	_nBufferIdx:= _nBufferIdx + 1;
	IF _nBufferIdx >= 3 THEN
		_nBufferIdx:= 1;
	END_IF

	CASE _nBufferIdx OF
		1:
			_pWriteBuffer:= _pBuffer1;
			_pReadBuffer:= _pBuffer2;

			_pWriteBufferTime:= ADR(_aBufferTime1);
			_pReadBufferTime:= ADR(_aBufferTime2);
		2:
			_pWriteBuffer:= _pBuffer2;
			_pReadBuffer:= _pBuffer1;

			_pWriteBufferTime:= ADR(_aBufferTime2);
			_pReadBufferTime:= ADR(_aBufferTime1);
	END_CASE

	nElements:= _nBufferEntry_Add;

	_nBufferEntry_Add:= 0;
	_bLock:= FALSE;
END_IF
END_METHOD

METHOD AddData : BOOL
VAR_INPUT
	pDataIn: PVOID;
END_VAR
VAR
END_VAR
IF TestAndSet(_bLock) THEN

	IF _pWriteBuffer <> 0 AND pDataIn <> 0 THEN

		IF _nBufferEntry_Add >= cEntryCount THEN
			_nBufferEntry_Add:= cEntryCount - 1;
		END_IF

		MEMCPY(_pWriteBuffer + (_nBufferEntry_Add * _nDataSize), pDataIn, _nDataSize);

		_nBufferEntry_Add:= _nBufferEntry_Add + 1;

		IF _pWriteBufferTime <> 0 THEN
			_pWriteBufferTime^[_nBufferEntry_Add]:= F_GetActualDcTime64();
		END_IF

	END_IF

	_bLock:= FALSE;
END_IF
END_METHOD

METHOD GetData : BOOL
VAR_INPUT
	nElement: UDINT(1..cEntryCount);
	pDataOut: PVOID;
END_VAR
VAR
END_VAR
IF nElement <= nElements THEN
	IF pDataOut <> 0 AND _pReadBuffer <> 0 THEN
		MEMCPY(pDataOut, _pReadBuffer + ((nElement-1) * _nDataSize), _nDataSize);
	END_IF
END_IF
END_METHOD

METHOD GetTimestamp : ULINT
VAR_INPUT
	nElement: UDINT(1..cEntryCount);
END_VAR
VAR
END_VAR
IF _pReadBufferTime <> 0 THEN
	GetTimestamp:= _pReadBufferTime^[nElement];
END_IF
END_METHOD

END_FUNCTION_BLOCK

// ---- POUs/Analytics/[Helper]/FB_GetSampleIndex.TcPOU
FUNCTION_BLOCK FB_GetSampleIndex
VAR_INPUT
	nSample: UDINT;
	nOverSamplingFactor: UDINT;
	nMaxOverSampling: UDINT;
	nTimestamp: ULINT;
END_VAR
VAR_OUTPUT
	bNewIndex: BOOL;
	nIndex: UDINT;
END_VAR
VAR
	nIndexFactor: UDINT;
	nLastIndex: UDINT;
	nLastTimestamp: ULINT;
END_VAR


nIndex:= 1;

IF nOverSamplingFactor > 0 THEN
	nIndexFactor:= nMaxOverSampling / nOverSamplingFactor;

	IF nIndexFactor > 0 THEN
		nIndex:= (nSample - 1) / nIndexFactor;
		nIndex:= nIndex + 1;
	END_IF

	IF nIndex > nOverSamplingFactor THEN
		nIndex:= nOverSamplingFactor;
	END_IF
END_IF

bNewIndex:= nIndex <> nLastIndex OR nLastTimestamp <> nTimestamp;

nLastIndex:= nIndex;
nLastTimestamp:= nTimestamp;

END_FUNCTION_BLOCK

// ---- POUs/Analytics/[Helper]/F_AlyTimestampToFileTime.TcPOU
FUNCTION F_AlyTimestampToFileTime : ULINT
VAR_INPUT
	tTimestamp: ULINT;
END_VAR
VAR
	tFileTime: T_FILETIME;
	
	fbToUTC: FB_TzSpecificLocalTimeToFileTime;
	//W. Europe Daylight Time
	//(UTC+01:00) Amsterdam, Berlin, Bern, Rome, Stockholm, Vienna
	tzInfo: ST_TimeZoneInformation := (bias := -60, standardDate := (wMonth := 10 ,wDay:=5, wHour := 3), daylightDate := (wMonth := 3, wDay:=5, wHour := 2), daylightBias := -60);
END_VAR

tFileTime:= DCTIME64_TO_Filetime(tTimestamp);

fbToUTC(in:= tFileTime, tzInfo:= tzInfo);
F_AlyTimestampToFileTime:= ULARGE_TO_ULINT(ULARGE_INTEGER(fbToUTC.out.dwHighDateTime, fbToUTC.out.dwLowDateTime));

END_FUNCTION

// ---- POUs/Analytics/[Helper]/F_AlyTimestampToLocalTime.TcPOU
FUNCTION F_AlyTimestampToLocalTime : ULINT
VAR_INPUT
	tTimestamp: ULINT;
END_VAR
VAR
	tFileTime: T_FILETIME;
END_VAR

tFileTime:= DCTIME64_TO_Filetime(tTimestamp);
F_AlyTimestampToLocalTime:= ULARGE_TO_ULINT(ULARGE_INTEGER(tFileTime.dwHighDateTime, tFileTime.dwLowDateTime));

END_FUNCTION

// ---- POUs/Analytics/[Helper]/F_ANY_Negation.TcPOU
FUNCTION F_ANY_Negation : BOOL
VAR_INPUT
	Input: ANY;
END_VAR
VAR
	bReturn: BOOL;
	pREAL: POINTER TO REAL;
	pLREAL: POINTER TO LREAL;
	pBOOL: POINTER TO BOOL;
	pBYTE: POINTER TO BYTE;
	pINT: POINTER TO INT;
	pDINT: POINTER TO DINT;
	pLINT: POINTER TO LINT;
	pUINT: POINTER TO UINT;
	pUDINT: POINTER TO UDINT;
	pULINT: POINTER TO ULINT;
	pWORD: POINTER TO WORD;
	pDWORD: POINTER TO DWORD;
	pLWORD: POINTER TO LWORD;
END_VAR

IF input.pValue <> 0 THEN
	bReturn:= TRUE;

	CASE Input.TypeClass OF
		__SYSTEM.TYPE_CLASS.TYPE_REAL:
			pREAL:= input.pValue;
			pREAL^:= pREAL^ * -1;
		__SYSTEM.TYPE_CLASS.TYPE_LREAL:
			pLREAL:= input.pValue;
			pLREAL^:= pLREAL^ * -1;
		__SYSTEM.TYPE_CLASS.TYPE_BOOL:
			pBOOL:= input.pValue;
			pBOOL^:= NOT pBOOL^;
		__SYSTEM.TYPE_CLASS.TYPE_BYTE:
			pBYTE:= input.pValue;
			pBYTE^:= NOT pBYTE^;
		__SYSTEM.TYPE_CLASS.TYPE_INT:
			pINT:= input.pValue;
			pINT^:= pINT^ * -1;
		__SYSTEM.TYPE_CLASS.TYPE_DINT:
			pDINT:= input.pValue;
			pDINT^:= pDINT^ * -1;
		__SYSTEM.TYPE_CLASS.TYPE_LINT:
			pLINT:= input.pValue;
			pLINT^:= pLINT^ * -1;
		__SYSTEM.TYPE_CLASS.TYPE_UINT:
			pUINT:= input.pValue;
			pUINT^:= NOT pUINT^;
		__SYSTEM.TYPE_CLASS.TYPE_UDINT:
			pUDINT:= input.pValue;
			pUDINT^:= NOT pUDINT^;
		__SYSTEM.TYPE_CLASS.TYPE_ULINT:
			pULINT:= input.pValue;
			pULINT^:= NOT pULINT^;
		__SYSTEM.TYPE_CLASS.TYPE_WORD:
			pWORD:= input.pValue;
			pWORD^:= NOT pWORD^;
		__SYSTEM.TYPE_CLASS.TYPE_DWORD:
			pDWORD:= input.pValue;
			pDWORD^:= NOT pDWORD^;
		__SYSTEM.TYPE_CLASS.TYPE_LWORD:
			pLWORD:= input.pValue;
			pLWORD^:= NOT pLWORD^;
		ELSE
			bReturn:= FALSE;
	END_CASE
END_IF

F_ANY_Negation:= bReturn;

END_FUNCTION

// ---- POUs/Analytics/[Helper]/F_ARRAY_To_LREAL_ARRAY.TcPOU
FUNCTION F_ARRAY_To_LREAL_ARRAY : BOOL
VAR_INPUT
	pDataIn: POINTER TO BYTE;
	cbDataIn: UDINT;
	eDataType: E_DTType;
END_VAR
VAR_IN_OUT
	aDataOut: ARRAY [*] OF LREAL;
END_VAR
VAR
	i: DINT;
	nPos: UDINT;
	
	pBOOL: POINTER TO BOOL;
	pBYTE: POINTER TO BYTE;
	pWORD: POINTER TO WORD;
	pDWORD: POINTER TO DWORD;
	pSINT: POINTER TO SINT;
	pUSINT: POINTER TO USINT;
	pINT: POINTER TO INT;
	pUINT: POINTER TO UINT;
	pDINT: POINTER TO DINT;
	pUDINT: POINTER TO UDINT;
	pLINT: POINTER TO LINT;
	pULINT: POINTER TO ULINT;
	pREAL: POINTER TO REAL;
	pLREAL: POINTER TO LREAL;
	pLWORD: POINTER TO LWORD;
END_VAR

FOR i := LOWER_BOUND(aDataOut,1) TO UPPER_BOUND(aDataOut,1) DO
	CASE eDataType OF
		E_DTType.NotInitialized:
			F_ARRAY_To_LREAL_ARRAY:= FALSE;
			RETURN;
		E_DTType.BOOL_:
			IF (nPos * 1) < cbDataIn THEN
				pBOOL:= pDataIn + (nPos * 1);
				aDataOut[i] := TO_LREAL(pBOOL^);
			END_IF
		E_DTType.BYTE_:
			IF (nPos * 1) < cbDataIn THEN
				pBYTE:= pDataIn + (nPos * 1);
				aDataOut[i] := TO_LREAL(pBYTE^);
			END_IF
		E_DTType.WORD_:
			IF (nPos * 2) < cbDataIn THEN
				pWORD:= pDataIn + (nPos * 2);
				aDataOut[i] := TO_LREAL(pWORD^);
			END_IF
		E_DTType.DWORD_:
			IF (nPos * 4) < cbDataIn THEN
				pDWORD:= pDataIn + (nPos * 4);
				aDataOut[i] := TO_LREAL(pDWORD^);
			END_IF
		E_DTType.SINT_:
			IF (nPos * 1) < cbDataIn THEN
				pSINT:= pDataIn + (nPos * 1);
				aDataOut[i] := TO_LREAL(pSINT^);
			END_IF
		E_DTType.INT_:
			IF (nPos * 2) < cbDataIn THEN
				pINT:= pDataIn + (nPos * 2);
				aDataOut[i] := TO_LREAL(pINT^);
			END_IF
		E_DTType.UINT_:
			IF (nPos * 2) < cbDataIn THEN
				pUINT:= pDataIn + (nPos * 2);
				aDataOut[i] := TO_LREAL(pUINT^);
			END_IF
		E_DTType.DINT_:
			IF (nPos * 4) < cbDataIn THEN
				pDINT:= pDataIn + (nPos * 4);
				aDataOut[i] := TO_LREAL(pDINT^);
			END_IF
		E_DTType.UDINT_:
			IF (nPos * 4) < cbDataIn THEN
				pUDINT:= pDataIn + (nPos * 4);
				aDataOut[i] := TO_LREAL(pUDINT^);
			END_IF
		E_DTType.LINT_:
			IF (nPos * 8) < cbDataIn THEN
				pLINT:= pDataIn + (nPos * 8);
				aDataOut[i] := TO_LREAL(pLINT^);
			END_IF
		E_DTType.ULINT_:
			IF (nPos * 8) < cbDataIn THEN
				pULINT:= pDataIn + (nPos * 8);
				aDataOut[i] := TO_LREAL(pULINT^);
			END_IF
		E_DTType.REAL_:
			IF (nPos * 4) < cbDataIn THEN
				pREAL:= pDataIn + (nPos * 4);
				aDataOut[i] := TO_LREAL(pREAL^);
			END_IF
		E_DTType.LREAL_:
			IF (nPos * 8) < cbDataIn THEN
				pLREAL:= pDataIn + (nPos * 8);
				aDataOut[i] := TO_LREAL(pLREAL^);
			END_IF
		E_DTType.LWORD_:
			IF (nPos * 8) < cbDataIn THEN
				pLWORD:= pDataIn + (nPos * 8);
				aDataOut[i] := TO_LREAL(pLWORD^);
			END_IF
	END_CASE

	nPos:= nPos + 1;
END_FOR

F_ARRAY_To_LREAL_ARRAY:= TRUE;

END_FUNCTION

// ---- POUs/Analytics/[Helper]/F_DCTimestructToFileTime.TcPOU
FUNCTION F_DCTimestructToFileTime : ULINT
VAR_INPUT
	dtTimestamp: DCTIMESTRUCT;
END_VAR
VAR
	dcTime: T_DCTIME64;
END_VAR

dcTime:= DCTIMESTRUCT_TO_DCTIME64(dtTimestamp);
F_DCTimestructToFileTime:= F_AlyTimestampToFileTime(dcTime);

END_FUNCTION

// ---- POUs/Analytics/[Helper]/F_FileTimeToDCTimestruct.TcPOU
FUNCTION F_FileTimeToDCTimestruct : DCTIMESTRUCT
VAR_INPUT
	tTimestamp: ULINT;
END_VAR
VAR
	tULarge: T_ULARGE_INTEGER;
	tFileTime: T_FILETIME;
	newDCTime: T_DCTIME64;
	
	fbToLocal: FB_FileTimeToTzSpecificLocalTime;
	//W. Europe Daylight Time
	//(UTC+01:00) Amsterdam, Berlin, Bern, Rome, Stockholm, Vienna
	tzInfo: ST_TimeZoneInformation := (bias := -60, standardDate := (wMonth := 10 ,wDay:=5, wHour := 3), daylightDate := (wMonth := 3, wDay:=5, wHour := 2), daylightBias := -60);
END_VAR

tULarge:= ULINT_TO_ULARGE(tTimestamp);
tFileTime.dwLowDateTime:= tULarge.dwLowPart;
tFileTime.dwHighDateTime:= tULarge.dwHighPart;

fbToLocal(in:= tFileTime, tzInfo:= tzInfo);
newDCTime:= FILETIME_TO_DCTIME64(fbToLocal.out);

F_FileTimeToDCTimestruct:= DCTIME64_TO_DCTIMESTRUCT(newDCTime);

END_FUNCTION

// ---- POUs/Analytics/[Helper]/F_SampleTimeCheck.TcPOU
FUNCTION F_SampleTimeCheck : BOOL
VAR_INPUT
	nSampleTimestamp: ULINT;
	nLastSampleTimestamp: ULINT;
	nSampleTime: UDINT;
END_VAR
VAR
	nDeviation: UDINT := 500000; //Allowed deviation 0.5ms
END_VAR

IF nLastSampleTimestamp = 0 THEN
	F_SampleTimeCheck:= TRUE;
ELSIF nSampleTimestamp >= (nLastSampleTimestamp + (nSampleTime + nDeviation)) THEN
	F_SampleTimeCheck:= TRUE;
ELSIF nSampleTimestamp >= (nLastSampleTimestamp + (nSampleTime - nDeviation)) THEN
	F_SampleTimeCheck:= TRUE;
ELSE
	F_SampleTimeCheck:= FALSE;
END_IF

END_FUNCTION

// ---- POUs/Analytics/[Helper]/F_ToANY.TcPOU
FUNCTION F_ToANY : __SYSTEM.AnyType
VAR_INPUT
	Input: ANY;
END_VAR
VAR
END_VAR

F_ToANY:= Input;

END_FUNCTION
